{attribute 'linkalways'} 
{attribute 'no_explicit_call' := 'This FB is a CLASS and must be accessed using methods or properties'}
{attribute 'enable_dynamic_creation'}
FUNCTION_BLOCK TestTwin EXTENDS BasicModbusDigitalTwin
VAR
	configData : TestSlaveConfigData;
	fastDataA : TestSlaveFastDataA;
	fastDataB : TestSlaveFastDataB;
	
	timeout : TIME := T#200MS;
END_VAR

{attribute 'monitoring' := 'call'}
PROPERTY PUBLIC Config1 : INT
GET // PUBLIC
Config1 := configData.config1;
END_GET
SET // PUBLIC
QueueWriteSingleRegister(0, INT_TO_WORD(Config1), timeout);
END_SET
END_PROPERTY

{attribute 'monitoring' := 'call'}
PROPERTY PUBLIC Config2 : INT
GET // PUBLIC
Config2 := configData.config2;
END_GET
SET // PUBLIC
QueueWriteSingleRegister(1, INT_TO_WORD(Config2), timeout);
END_SET
END_PROPERTY

{attribute 'monitoring' := 'call'}
PROPERTY PUBLIC Data1 : INT
GET // PUBLIC
Data1 := fastDataA.fastData1;
END_GET
SET // PUBLIC
QueueWriteSingleRegister(2, INT_TO_WORD(Data1), timeout);
END_SET
END_PROPERTY

{attribute 'monitoring' := 'call'}
PROPERTY PUBLIC Data2 : INT
GET // PUBLIC
Data2 := fastDataA.fastData2;
END_GET
SET // PUBLIC
QueueWriteSingleRegister(3, INT_TO_WORD(Data2), timeout);
END_SET
END_PROPERTY

{attribute 'monitoring' := 'call'}
PROPERTY PUBLIC Data3 : INT
GET // PUBLIC
Data3 := fastDataB.fastData3;
END_GET
SET // PUBLIC
QueueWriteSingleRegister(4, INT_TO_WORD(Data3), timeout);
END_SET
END_PROPERTY

{attribute 'monitoring' := 'call'}
PROPERTY PUBLIC Data4 : INT
GET // PUBLIC
Data4 := fastDataB.fastData4;
END_GET
SET // PUBLIC
QueueWriteSingleRegister(5, INT_TO_WORD(Data4), timeout);
END_SET
END_PROPERTY

METHOD FB_init : BOOL
VAR_INPUT
	bInitRetains : BOOL; // if TRUE, the retain variables are initialized (warm start / cold start)
	bInCopyCode : BOOL;  // if TRUE, the instance afterwards gets moved into the copy code (online change)
	ipAddress : STRING(15);
	tcpPort : UINT := MODBUS_TCP_PORT;
	unitId : USINT;
END_VAR
AddCyclicalReadRegisters(0, 2, ADR(configData), SIZEOF(configData), timeout);
AddCyclicalReadRegisters(2, 2, ADR(fastDataA), SIZEOF(fastDataA), timeout);
AddCyclicalReadRegisters(4, 2, ADR(fastDataB), SIZEOF(fastDataB), timeout);
END_METHOD

END_FUNCTION_BLOCK

(* stored: Version 1.1.0.1, ProductVersion 3.1.4024.12
   POU TestTwin: Id {560363cb-337e-4204-b176-aa17769a2df9}, SpecialFunc None
   Folder Properties: Id {1d00b0d0-d8f9-49c6-8596-4ed75dbf6670}
   Property Config1: Id {3d612441-b9a2-43d9-96ab-a8fd0b5862a5}
   Get Get: Id {0411bcfc-d280-4a2f-b31b-3e12a94eb2b4}
   Set Set: Id {041da7b9-b29a-4753-9b76-510e5dafc800}
   Property Config2: Id {427d1ae4-a56f-444d-92a2-9813240e331e}
   Get Get: Id {f7ec2980-ac93-4f9d-a0ea-6fc8775d07e5}
   Set Set: Id {320c12a2-e007-44b0-9422-eb7dfa155d72}
   Property Data1: Id {4cd4f67a-5e98-4718-974c-248691edd2f5}
   Get Get: Id {b6183a83-5567-4b06-8958-fd524c598ac8}
   Set Set: Id {0a3d8920-7061-4b48-8f61-389c2d4761b4}
   Property Data2: Id {c500f905-27f7-4e2d-aea3-555279887e74}
   Get Get: Id {0e17e688-dd3d-4202-995f-9468f5199a1e}
   Set Set: Id {906ef892-3ff3-408e-b0f3-260f11b7e4f6}
   Property Data3: Id {cedcc904-47d2-46b2-918a-aebd2b843aed}
   Get Get: Id {c5b83bdc-60ef-4415-9c7a-508e6d9287e1}
   Set Set: Id {c2303dfc-0f01-4fe8-bc18-95f4c93ea39d}
   Property Data4: Id {ac7da84c-02b5-4f40-99ee-568bf6e6b1d6}
   Get Get: Id {7b50e30b-ff4a-435d-9ec4-a3d9fb51e2e9}
   Set Set: Id {ad906674-c446-4c51-ba85-40e32e0f146d}
   Method FB_init: Id {91f685b6-9577-43b7-961f-9ebd7adaf0da} *)
